FUNCTION_BLOCK L3_SendPart (* Basic Function Block Type *)
  (* Standard: 61499-2 *)
  (* Version 0.0, 2014-10-02, EQUEROL, UJI *)
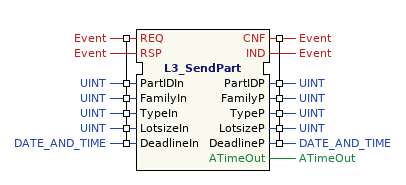
  EVENT_INPUT
    REQ WITH PartIDIn, FamilyIn, TypeIn, LotsizeIn, DeadlineIn; (* Normal Execution Request *)
    RSP; (* Response indicating the correct reception of the order *)
  END_EVENT
  EVENT_OUTPUT
    CNF WITH PartIDP, FamilyP, TypeP, LotsizeP, DeadlineP; (* Execution Confirmation *)
    IND; (* Indication of efectively sent order *)
  END_EVENT
  VAR_INPUT
    PartIDIn : UINT; (* Part's identifier *)
    FamilyIn : UINT; (* Part's family *)
    TypeIn : UINT; (* Part's type *)
    LotsizeIn : UINT; (* Number of parts to be manufactured *)
    DeadlineIn : DATE_AND_TIME; (* Order deadline *)
  END_VAR
  VAR_OUTPUT
    PartIDP : UINT; (* Part's identifier *)
    FamilyP : UINT; (* Part's family *)
    TypeP : UINT; (* Part's type *)
    LotsizeP : UINT; (* Number of parts to be manufatured *)
    DeadlineP : DATE_AND_TIME; (* Order deadline *)
  END_VAR
  PLUGS
    ATimeOut : ATimeOut;
  END_PLUGS
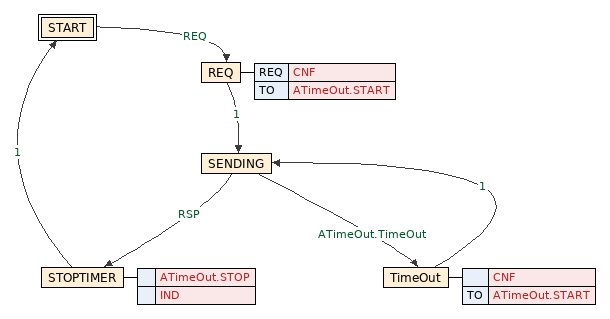
  EC_STATES
    START; (* Initial State *)
    REQ : REQ -> CNF, TO -> ATimeOut.START; (* Normal execution *)
    SENDING;
    TimeOut : -> CNF, TO -> ATimeOut.START;
    STOPTIMER : -> ATimeOut.STOP, -> IND;
  END_STATES
  EC_TRANSITIONS
    START TO REQ := REQ;
    REQ TO SENDING := 1;
    SENDING TO TimeOut := ATimeOut.TimeOut;
    SENDING TO STOPTIMER := RSP;
    STOPTIMER TO START := 1;
    TimeOut TO SENDING := 1;
  END_TRANSITIONS
  ALGORITHM REQ IN ST: (* Normally executed algorithm *)
PartIDP := PartIDIn;
FamilyP := FamilyIn;
TypeP := TypeIn;
LotsizeP := LotsizeIn;
DeadlineP := DeadlineIn;
  END_ALGORITHM
  ALGORITHM TO IN ST: (* new algorithm *)
ATimeOut.DT := TIME#1000ms;
  END_ALGORITHM
END_FUNCTION_BLOCK
